// TIA Portal V21 export
VAR_GLOBAL   // PLC tag table "K_SezioniPastorizzatore"
END_VAR
VAR_GLOBAL CONSTANT   // user constants
   K_SezionePastorizzatore_Sez1 : Int := 1;
   K_SezionePastorizzatore_Sez2 : Int := 2;
   K_SezionePastorizzatore_Sez3 : Int := 3;
   K_SezionePastorizzatore_Sez4 : Int := 4;
   K_SezionePastorizzatore_Sez5 : Int := 5;
   K_SezionePastorizzatore_Sez6 : Int := 6;
   K_SezionePastorizzatore_Sez7 : Int := 7;
   K_SezionePastorizzatore_Sez8 : Int := 8;
   K_SezionePastorizzatore_Sez9 : Int := 9;
   K_SezionePastorizzatore_Sez10 : Int := 10;
END_VAR
